	bTrackBuild		: BOOL;
	StartFromTrack	: I_Track;
	EndAtTrack		: I_Track;
END_VAR
fbR_TrigExecute(CLK := bExecute);
IF fbR_TrigExecute.Q AND NOT bBusy THEN
	nState := 10;
	bBusy := TRUE;
	bError := FALSE;
END_IF


CASE nState OF 

	10:	// Init Track-Table
	
		// *******************************************************************
		// *** This code must be eddited according to machine/track layout ***
		// *******************************************************************
	
		nStartFromTrack	:= 0;		// 0 for the first track all others according to their predecessor!
	    	nEndAtTrack := 0;		// 0 for the first track all others according to their successor! 		
		     bCloseLoop := FALSE;	// TRUE for circular track	
			
			
		TrackTable[1,1] :=   0.0;	// x-koordinate
		TrackTable[1,2] :=   0.0;	// y-koordinate
		TrackTable[1,3] :=   0.0;	// c
		
		TrackTable[2,1] :=   0.0;	// x-koordinate
		TrackTable[2,2] :=   0.0;	// y-koordinate
		TrackTable[2,3] :=   0.0;	// c		
		
		TrackTable[3,1] :=   0.0;	// x-koordinate
		TrackTable[3,2] :=   0.0;	// y-koordinate
		TrackTable[3,3] :=   0.0;	// c		
	
		TrackTable[4,1] :=   0.0;	// x-koordinate
		TrackTable[4,2] :=   0.0;	// y-koordinate
		TrackTable[4,3] :=   0.0;	// c		
	
		TrackTable[5,1] :=   0.0;	// x-koordinate
		TrackTable[5,2] :=   0.0;	// y-koordinate
		TrackTable[5,3] :=   0.0;	// c		
	
		TrackTable[6,1] :=   0.0;	// x-koordinate
		TrackTable[6,2] :=   0.0;	// y-koordinate
		TrackTable[6,3] :=   0.0;	// c				
		
		nState := 20;
		
		
	20:	// Building the track
		IF nStartFromTrack > 0 THEN
			StartFromTrack := ipTrack[nStartFromTrack];
		END_IF
		
		IF nEndAtTrack > 0 THEN
			EndAtTrack := ipTrack[nStartFromTrack];
		END_IF

		bTrackBuild := FALSE;
		IF  nStartFromTrack > 0 
		AND     nEndAtTrack > 0
		THEN
			IF fbTrackStandard.BuildTrack(TrackTable, StartFromTrack.std, EndAtTrack.std, bCloseLoop) THEN
				bTrackBuild := TRUE;
			END_IF
		ELSIF nStartFromTrack > 0 THEN
			IF fbTrackStandard.BuildTrack(TrackTable, StartFromTrack.std, 0, bCloseLoop) THEN
				bTrackBuild := TRUE;
			END_IF
		ELSIF nEndAtTrack > 0 THEN
			IF fbTrackStandard.BuildTrack(TrackTable, 0, EndAtTrack.std, bCloseLoop) THEN
				bTrackBuild := TRUE;
			END_IF
		ELSE
			IF fbTrackStandard.BuildTrack(TrackTable, 0, 0, bCloseLoop) THEN
				bTrackBuild := TRUE;
			END_IF			
		END_IF
		
		IF bTrackBuild THEN
			nState := 30;	
		END_IF
	
		
	30: 	
		IF fbTrackStandard.P_BuildTrack.Done THEN
			nState := 100;
		END_IF
		
					 
	100: 	// Track build done
			fTrackLength := fbTrackStandard.GetLength();
				   bBusy := FALSE;
			  Initialize := TRUE;
			
			IF NOT bExecute THEN
				Initialize := FALSE;
				    nState := 0;
			END_IF
	
END_CASE
END_METHOD

END_FUNCTION_BLOCK

// ---- 1_Industry/VISUs/OperationalControlPad.TcVIS
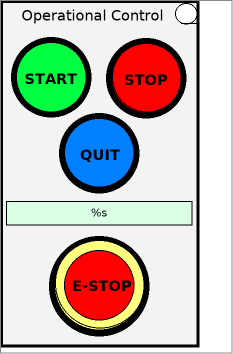
VISUALIZATION OperationalControlPad  // 233x354
VAR_IN_OUT
	stVisOperationalControl	: ST_Vis_OperationalControl;
END_VAR
    Rectangle (0,0 199x347)
    Label (9,1 167x29), "Operational Control"
    Ellipse (11,37 80x80)
    Ellipse (16,42 70x70)
    Ellipse (16,42 70x70), invisible if: NOT stVisOperationalControl.bStartButtonLamp
    Ellipse (106,38 80x80)
    Ellipse (111,43 70x70)
    Ellipse (111,43 70x70), invisible if: Not stVisOperationalControl.bStopButtonLamp
    Ellipse (59,113 80x80)
    Ellipse (64,118 70x70)
    Ellipse (64,118 70x70), invisible if: NOT stVisOperationalControl.bQuitButtonLamp
    Label (13,64 76x30), "START"
    Label (108,65 76x30), "STOP"
    Label (62,140 76x30), "QUIT"
    Rectangle (6,201 186x24), "%s", text variable: stVisOperationalControl.sMessage
    Ellipse (49,236 100x100)
    Ellipse (54,240 90x90)
    Ellipse (64,250 70x70)
    Ellipse (64,250 70x70), invisible if: NOT stVisOperationalControl.bEStopButtonLamp
    Label (64,271 76x30), "E-STOP"
    Rectangle (6,201 186x24), "%s", text variable: stVisOperationalControl.sMessage, invisible if: NOT stVisOperationalControl.bMessageColorRed
    Rectangle (6,201 186x24), "%s", text variable: stVisOperationalControl.sMessage, invisible if: NOT stVisOperationalControl.bMessageColorGreen
    Ellipse (16,42 70x70)
        tap stVisOperationalControl.bStartButtunState
    Ellipse (112,42 70x70)
        tap stVisOperationalControl.bStopButtonState
    Ellipse (64,117 70x70)
        tap stVisOperationalControl.bQuitButtonState
    Ellipse (55,238 90x90)
        toggle stVisOperationalControl.bEStopButtonState
    Ellipse (175,3 22x21)
    Line (218,-7) (233,-6)
    Line (181,23) (197,23)
    Rectangle (158,2 40x30)
        OnMouseClick: execute { stVisOperationalControl.bVisInvisibleButton := TRUE; }
END_VISUALIZATION

// ---- 1_Industry/VISUs/StarterKitStateMachinelPad.TcVIS
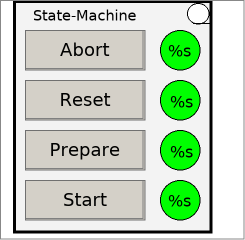
VISUALIZATION StarterKitStateMachinelPad  // 245x240
VAR_IN_OUT
	
	stControlPadControl		:   ST_Vis_ControlPadControl;

END_VAR
    Rectangle (13,0 199x233)
    Button (25,30 120x40), "Abort"
        tap stControlPadControl.bButtonState_Abort p3779583253=TRUE
    Button (25,80 120x40), "Reset"
        tap stControlPadControl.bButtonState_Reset
    Button (25,130 120x40), "Prepare"
        tap stControlPadControl.bButtonState_Prepare
    Button (25,180 120x40), "Start"
        tap stControlPadControl.bButtonState_Start
    Ellipse (160,30 40x40)
    Ellipse (160,30 40x40), invisible if: NOT stControlPadControl.bStateSignalAbortYellow
    Group (160,80 40x40)
        Ellipse (0,0 40x40)
        Ellipse (0,0 40x40), invisible if: NOT stControlPadControl.bStateSignalResetYellow
        Ellipse (0,0 40x40), invisible if: NOT stControlPadControl.bStateSignalResetGreen
    Group (160,130 40x40)
        Ellipse (0,0 40x40)
        Ellipse (0,0 40x40), invisible if: NOT stControlPadControl.bStateSignalPrepareYellow
        Ellipse (0,0 40x40), invisible if: NOT stControlPadControl.bStateSignalPrepareGreen
    Group (160,180 40x40)
        Ellipse (0,0 40x40)
        Ellipse (0,0 40x40), invisible if: NOT stControlPadControl.bStateSignalExecuteYellow
        Ellipse (0,0 40x40), invisible if: NOT stControlPadControl.bStateSignalExecuteGreen
    Ellipse (160,30 40x40), invisible if: NOT stControlPadControl.bStateSignalAbortBlue
    Ellipse (160,30 40x40), invisible if: NOT stControlPadControl.bStateSignalAbortGreen
    Label (19,1 132x29), "State-Machine"
    Textfield (159,35 42x32), "%s", text variable: stControlPadControl.iAbortSequenceState, invisible if: stControlPadControl.bAbortSequenceStateInvisible
    Textfield (161,86 42x32), "%s", text variable: stControlPadControl.iResetSequenceState, invisible if: stControlPadControl.bResetSequenceStateInvisible
    Textfield (161,136 42x32), "%s", text variable: stControlPadControl.iPrepareSequenceState, invisible if: stControlPadControl.bPrepareSequenceStateInvisible
    Textfield (159,185 42x32), "%s", text variable: stControlPadControl.iStartSequenceState, invisible if: stControlPadControl.bStartSequenceStateInvisible
    Ellipse (187,3 22x21)
    Line (230,-7) (245,-6)
    Line (193,23) (209,23)
    Rectangle (179,3 32x25)
        OnMouseClick: execute { stControlPadControl.bVisInvisibleButton := TRUE; }
END_VISUALIZATION

// ---- GlobalTextList.TcGTLO
TEXTLIST GlobalTextList
  632 = '\txPlanar'
  135 = '\tXPlanar'
  427 = '\nGroup\nNotReady'
  425 = '\nGroup\nStandby'
  140 = '%.3f'
  243 = '%d'
  602 = '%d /'
  145 = '%d Axes'
  43 = '%s'
  245 = '+'
  246 = '-'
  532 = '/'
  81 = '1'
  902 = '2'
  489 = '3'
  115 = '4'
  268 = '5'
  274 = 'A'
  39 = 'Abort'
  56 = 'Activated'
  726 = 'Activating'
  774 = 'ActivationState'
  215 = 'B'
  306 = 'Busy'
  671 = 'C'
  224 = 'CA_Group'
  560 = 'E-STOP'
  144 = 'Enable Requested FALSE'
  143 = 'Enable Requested TRUE'
  51 = 'Entrance Location'
  790 = 'Error in the Group or in one of the axes'
  789 = 'error on the\ngroup or in one\nof the axes'
  331 = 'Error: %d'
  1811 = 'Exit Location'
  146 = 'General'
  431 = 'Group\nErrorDisabled'
  430 = 'Group\nErrorEnabled'
  429 = 'GroupDisabled'
  428 = 'GroupErrorStop'
  424 = 'GroupMoving'
  426 = 'GroupStopping'
  750 = 'GVL_StationVisu.aMoverInQueue[INDEX]'
  748 = 'GVL_StationVisu.aMoverInSequence[INDEX].nMover'
  749 = 'GVL_StationVisu.aMoverInSequence[INDEX].nSequence'
  413 = 'GVL_XPlanarVisuDiag.aMoverInSequence[INDEX].nMover'
  498 = 'GVL_XPlanarVisuDiag.aMoverInSequence[INDEX].nSequence'
  53 = 'Home'
  152 = 'Inactive'
  142 = 'INVALID'
  938 = 'M1'
  303 = 'M2'
  38 = 'M3'
  609 = 'M4'
  432 = 'MC_AddAxis'
  783 = 'MC_GroupDisable'
  786 = 'MC_GroupEnable'
  784 = 'MC_GroupHalt'
  434 = 'MC_GroupReset'
  785 = 'MC_GroupStop'
  433 = 'MC_RemAxis'
  787 = 'MC_UngroupAllAxes'
  114 = 'Mover'
  348 = 'Mover:'
  522 = 'MoverId:'
  1100 = 'NumMoversReq.'
  788 = 'one axis\nnot ready'
  807 = 'OnTrack'
  105 = 'Operational Control'
  49 = 'Operational Control Pad'
  819 = 'PosA'
  255 = 'PosB'
  653 = 'PosC'
  837 = 'PosX'
  932 = 'PosY'
  30 = 'PosZ'
  953 = 'Prepare'
  927 = 'Process'
  1737 = 'Prozess Location'
  1111 = 'Queue'
  872 = 'Queue Location'
  509 = 'QueueGap'
  675 = 'QueuePositions'
  134 = 'QUIT'
  40 = 'Reset'
  42 = 'Run'
  41 = 'Start'
  678 = 'START'
  260 = 'State'
  390 = 'State-Machine'
  839 = 'State-Machine Pad'
  291 = 'Station'
  197 = 'Station Parameter'
  461 = 'Station: %d'
  1657 = 'Station: %s'
  141 = 'Status'
  939 = 'STOP'
  499 = 'Track'
  900 = 'X'
  313 = 'y'
END_TEXTLIST

// ---- VISUs/CmdHistory/VI_CmdHistorySide.TcVIS
VISUALIZATION VI_CmdHistorySide  // 2x2
END_VISUALIZATION

// ---- VISUs/CmdHistory/VI_CmdHistorySub.TcVIS
VISUALIZATION VI_CmdHistorySub  // 2x2
END_VISUALIZATION

// ---- VISUs/ControlXplanar/VI_Control_Xplanar.TcVIS
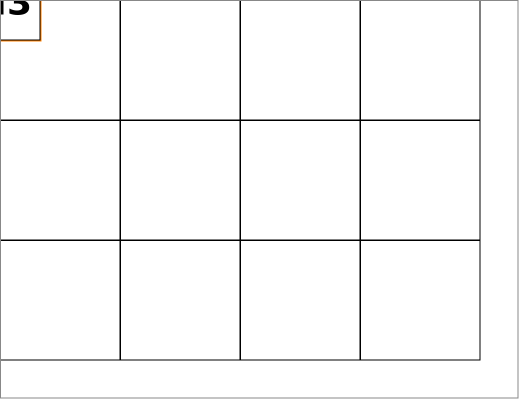
VISUALIZATION VI_Control_Xplanar  // 519x399
    Rectangle (0,0 120x120)
    Rectangle (120,0 120x120)
    Rectangle (240,0 120x120)
    Rectangle (360,0 120x120)
    Rectangle (0,120 120x120)
    Rectangle (120,120 120x120)
    Rectangle (240,120 120x120)
    Rectangle (360,120 120x120)
    Rectangle (0,240 120x120)
    Rectangle (120,240 120x120)
    Rectangle (240,240 120x120)
    Rectangle (360,240 120x120)
    Rectangle (-39,-39 80x80), "1"
        p3560616238: MAIN.fbXMotionUnit.fbStation_01_Process.VisuPosX/2
        p2738717112: (720-MAIN.fbXMotionUnit.fbStation_01_Process.VisuPosY)/2
    Rectangle (-39,-39 80x80), "2"
        p3560616238: MAIN.fbXMotionUnit.fbStation_02_Process.VisuPosX/2
        p2738717112: (720-MAIN.fbXMotionUnit.fbStation_02_Process.VisuPosY)/2
    Rectangle (-39,-39 80x80), "3"
        p3560616238: MAIN.fbXMotionUnit.fbStation_03_Process.VisuPosX/2
        p2738717112: (720-MAIN.fbXMotionUnit.fbStation_03_Process.VisuPosY)/2
    Rectangle (-39,-39 80x80), "4"
        p3560616238: MAIN.fbXMotionUnit.fbStation_04_Switch.VisuPosX/2
        p2738717112: (720-MAIN.fbXMotionUnit.fbStation_04_Switch.VisuPosY)/2
    Rectangle (-39,-39 80x80), "5"
        p3560616238: MAIN.fbXMotionUnit.fbStation_05_Switch.VisuPosX/2
        p2738717112: (720-MAIN.fbXMotionUnit.fbStation_05_Switch.VisuPosY)/2
    Rectangle (-37,-37 77x77), "M1"
        p3560616238: MAIN.fbXMotionUnit.fbMover[1].VisuPos.x/2
        p2738717112: (720-MAIN.fbXMotionUnit.fbMover[1].VisuPos.y)/2
    Rectangle (-37,-37 77x77), "M2"
        p3560616238: MAIN.fbXMotionUnit.fbMover[2].VisuPos.x/2
        p2738717112: (720-MAIN.fbXMotionUnit.fbMover[2].VisuPos.y)/2
    Rectangle (-37,-37 77x77), "M4"
        p3560616238: MAIN.fbXMotionUnit.fbMover[4].VisuPos.x/2
        p2738717112: (720-MAIN.fbXMotionUnit.fbMover[4].VisuPos.y)/2
    Rectangle (-37,-37 77x77), "M3"
        p3560616238: MAIN.fbXMotionUnit.fbMover[3].VisuPos.x/2
        p2738717112: (720-MAIN.fbXMotionUnit.fbMover[3].VisuPos.y)/2
END_VISUALIZATION

// ---- VISUs/Helper/VI_NumberHollow.TcVIS
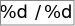
VISUALIZATION VI_NumberHollow  // 75x26
VAR_IN_OUT
	nNumberToDisplay : INT;
	nMaxNumberToDisplay : INT;
END_VAR
    Rectangle (-3,0 34x24), "%d", text variable: nNumberToDisplay
    Rectangle (41,0 32x24), "%d", text variable: nMaxNumberToDisplay
    Rectangle (27,0 17x24), "/", text variable: GVL_XtsVisuLib.nXtsIdMaxToDisplay
END_VISUALIZATION

// ---- VISUs/Helper/VI_NumberSub.TcVIS
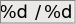
VISUALIZATION VI_NumberSub  // 76x24
VAR_IN_OUT
	nNumberToDisplay : INT;
	nMaxNumberToDisplay : INT;
END_VAR
    Rectangle (-3,0 34x24), "%d", text variable: nNumberToDisplay
    Rectangle (41,0 32x24), "%d", text variable: nMaxNumberToDisplay
    Rectangle (27,0 17x24), "/"
END_VISUALIZATION

// ---- VISUs/Station/VI_Station.TcVIS
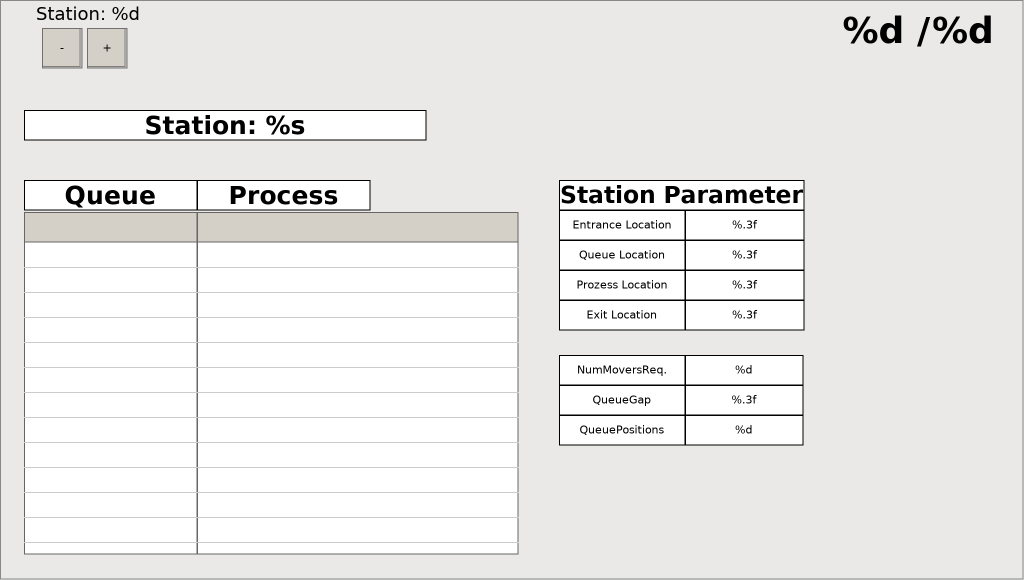
VISUALIZATION VI_Station  // 1024x580
    Frame (0,80 1024x500)
        shows VI_StationSub()
    Rectangle (929,5 77x51), "%d", text variable: GVL_XPlanarVisuDiag.nMaxStationToDisplay
    Rectangle (830,5 103x51), "%d /", text variable: GVL_XPlanarVisuDiag.nStationIdToDisplay
    Button (87,28 40x40), "+", invisible if: GVL_StationVisu.bStationNextInvisible
        tap GVL_XPlanarVisuDiag.bStationNext p1329445385=TRUE
    Button (42,28 40x40), "-", invisible if: GVL_XPlanarVisuDiag.bSationPreviousInvisible
        tap GVL_XPlanarVisuDiag.bStationPrevious
    Rectangle (34,2 108x24), "Station: %d", text variable: GVL_XPlanarVisuDiag.nStationIdToDisplay
END_VISUALIZATION

// ---- VISUs/Station/VI_StationSub.TcVIS
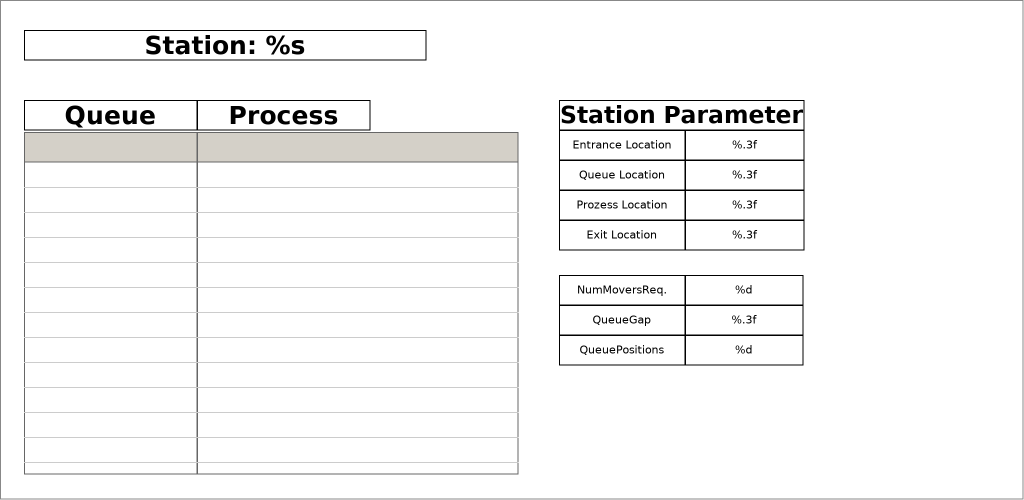
VISUALIZATION VI_StationSub  // 1024x500
    Rectangle (24,30 402x30), "Station: %s", text variable: GVL_XPlanarVisuDiag.sStationName
    Rectangle (24,100 173x30), "Queue"
    Rectangle (197,100 173x30), "Process"
    Table (197,132 321x342), data array: GVL_StationVisu.aMoverInSequence
        p1128707560: GVL_XPlanarVisuDiag.gcnMaxMoverInStation
        p3854506369: GVL_StationVisu.aMoverInSequence[INDEX].nMover
        p1892666644: GVL_StationVisu.aMoverInSequence[INDEX].nSequence
        p2232123230: GVL_XPlanarVisuDiag.aMoverInSequence[INDEX].nMover
        p511219082: GVL_XPlanarVisuDiag.aMoverInSequence[INDEX].nSequence
    Table (24,132 173x342), data array: GVL_XPlanarVisuDiag.aMoverInQueue
        p1128707560: GVL_XPlanarVisuDiag.gcnMaxMoverInStation
        p3854506369: GVL_XPlanarVisuDiag.aMoverInQueue[INDEX]
    Rectangle (559,100 245x30), "Station Parameter"
    Rectangle (559,130 126x30), "Entrance Location"
    Rectangle (559,160 126x30), "Queue Location"
    Rectangle (559,190 126x30), "Prozess Location"
    Rectangle (559,220 126x30), "Exit Location"
    Rectangle (559,275 126x30), "NumMoversReq."
    Rectangle (559,305 126x30), "QueueGap"
    Rectangle (559,335 126x30), "QueuePositions"
    Rectangle (685,130 119x30), "%.3f", text variable: GVL_XPlanarVisuDiag.stStationConfig.fEntranceLocation
    Rectangle (685,160 119x30), "%.3f", text variable: GVL_XPlanarVisuDiag.stStationConfig.fQueueLocation
    Rectangle (685,190 119x30), "%.3f", text variable: GVL_XPlanarVisuDiag.stStationConfig.fProzessLocation
    Rectangle (685,220 119x30), "%.3f", text variable: GVL_XPlanarVisuDiag.stStationConfig.fExitLocation
    Rectangle (685,275 118x30), "%d", text variable: GVL_XPlanarVisuDiag.stStationConfig.nNumMoversRequired
    Rectangle (685,305 118x30), "%.3f", text variable: GVL_XPlanarVisuDiag.stStationConfig.fQueueGap
    Rectangle (685,335 118x30), "%d", text variable: GVL_XPlanarVisuDiag.stStationConfig.nNumQueuePositions
END_VISUALIZATION

// ---- VISUs/Visualization.TcVIS
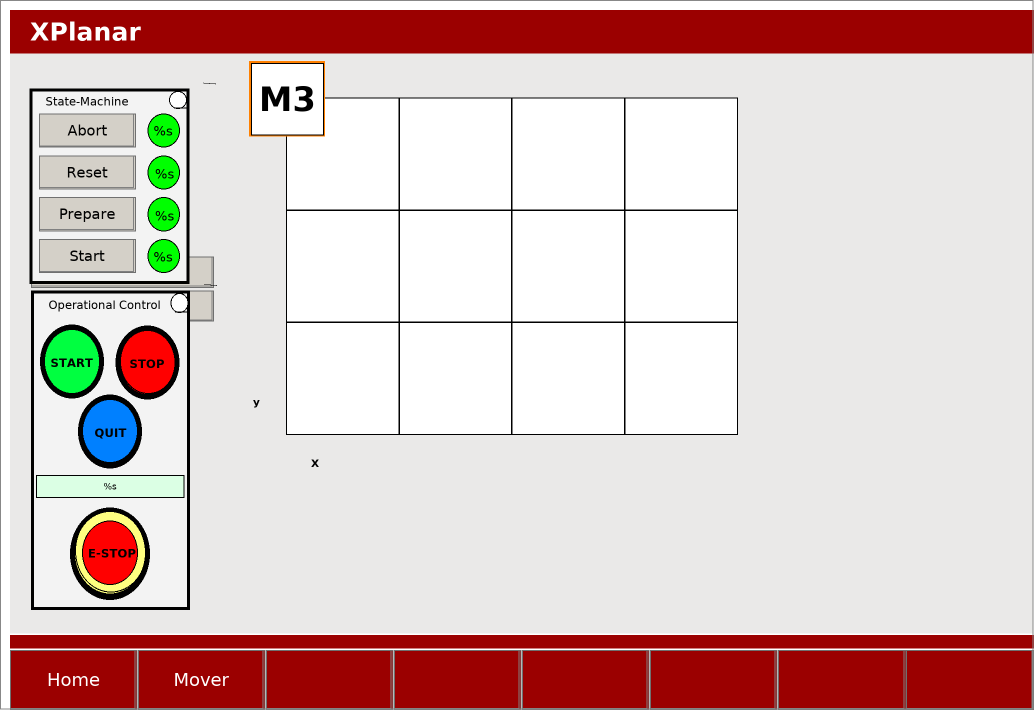
VISUALIZATION Visualization  // 1034x710
    Frame (10,53 1023x580)
        shows VI_MainSide()
        shows Tc3_XPlanarStandard.VI_MoverLogOverview()
        shows VI_EtherCatDiag()
        shows VI_MoverDiag()
        shows VI_MoverTuning()
        shows VI_MoverDiag()
        shows VI_Station()
        p1165984742: GVL_XtsVisu.pGroupRef[1]^.NcToPlc.Common.GroupStatus
        p547225198: GVL_XtsVisu.pGroupRef[1]
    Rectangle (10,10 1024x43), "XPlanar"
    Rectangle (10,635 1024x13)
    Button (10,650 127x60), "Home"
        OnMouseDown: FrameSelectionChange Selection=SelectedFrame=87eec691-4479-469a-bdd2-91ec7a1bb6bd, GlobSel=AssignType=Directly, SelType=Locally
    Button (138,650 127x60), "Mover"
        OnMouseUp: FrameSelectionChange Selection=SelectedFrame=87eec691-4479-469a-bdd2-91ec7a1bb6bd, Selection=1, GlobSel=AssignType=Directly, SelType=Locally
    Button (266,650 127x60)
    Button (394,650 127x60)
    Button (522,650 127x60)
    Button (650,650 127x60)
    Button (906,650 128x60)
    Button (778,650 128x60)
END_VISUALIZATION

// ---- VISUs/Visualization.TcVIS
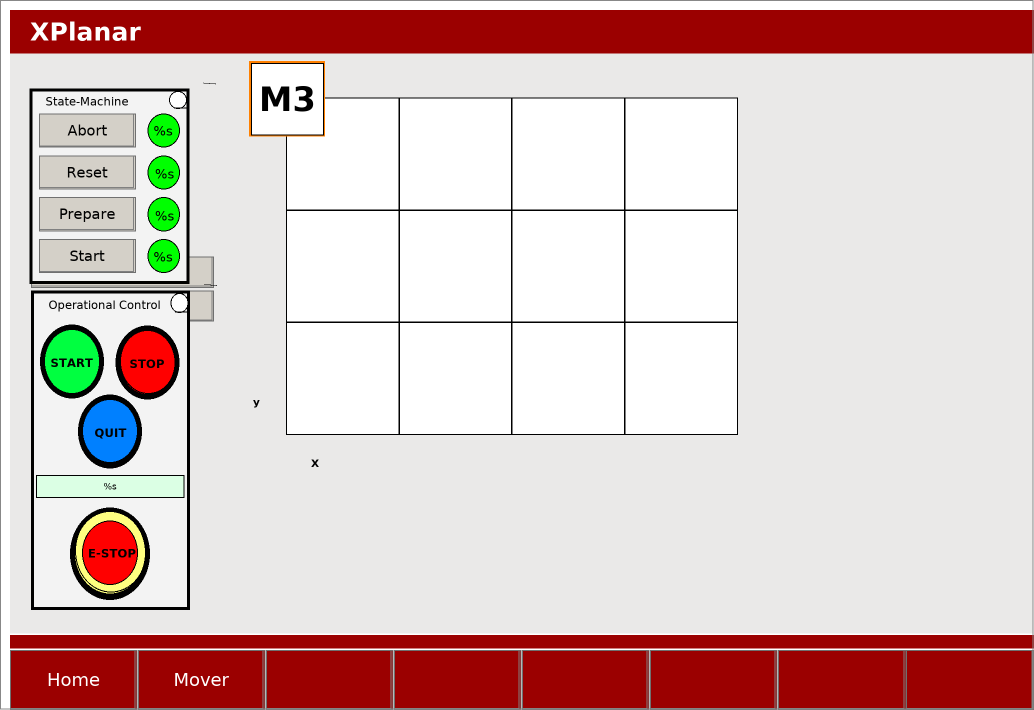
VISUALIZATION Visualization  // 1034x710
    Frame (10,53 1023x580)
        shows VI_MainSide()
        shows Tc3_XPlanarStandard.VI_MoverLogOverview()
        shows VI_EtherCatDiag()
        shows VI_MoverDiag()
        shows VI_MoverTuning()
        shows VI_MoverDiag()
        shows VI_Station()
        p1165984742: GVL_XtsVisu.pGroupRef[1]^.NcToPlc.Common.GroupStatus
        p547225198: GVL_XtsVisu.pGroupRef[1]
    Rectangle (10,10 1024x43), "XPlanar"
    Rectangle (10,635 1024x13)
    Button (10,650 127x60), "Home"
        OnMouseDown: FrameSelectionChange Selection=SelectedFrame=87eec691-4479-469a-bdd2-91ec7a1bb6bd, GlobSel=AssignType=Directly, SelType=Locally
    Button (138,650 127x60), "Mover"
        OnMouseUp: FrameSelectionChange Selection=SelectedFrame=87eec691-4479-469a-bdd2-91ec7a1bb6bd, Selection=1, GlobSel=AssignType=Directly, SelType=Locally
    Button (266,650 127x60)
    Button (394,650 127x60)
    Button (522,650 127x60)
    Button (650,650 127x60)
    Button (906,650 128x60)
    Button (778,650 128x60)
END_VISUALIZATION

// ---- VISUs/VI_MainSide.TcVIS
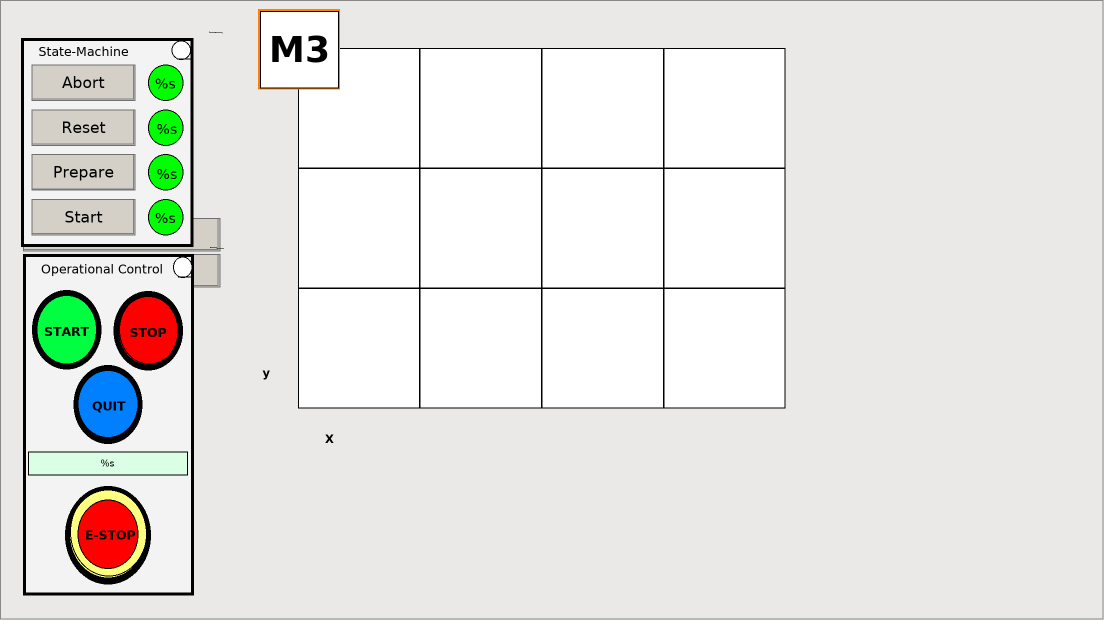
VISUALIZATION VI_MainSide  // 1104x620
    Polygon (172,343) (173,344)
    Frame (298,48 527x399)
        shows VI_Control_Xplanar()
    Label (316,424 27x30), "X"
    Label (253,358 27x30), "y"
    Button (23,254 197x33), "Operational Control Pad", invisible if: NOT stVisControl.stOperatorPad.bVisInvisible
        p3560616238: stVisControl.stOperatorPad.nButtonPositionX
        p2738717112: stVisControl.stOperatorPad.nButtonPositionY
        OnMouseClick: execute { stVisControl.stOperatorPad.bVisInvisibleButton := FALSE; }
    Button (23,218 197x33), "State-Machine Pad", invisible if: NOT stVisControl.stControlPad.bVisInvisible
        p3560616238: stVisControl.stControlPad.nButtonPositionX
        p2738717112: stVisControl.stControlPad.nButtonPositionY
        OnMouseClick: execute { stVisControl.stControlPad.bVisInvisibleButton := FALSE; }
    Frame (10,38 212x215), invisible if: stVisControl.stControlPad.bVisInvisible
        shows StarterKitStateMachinelPad(stControlPadControl := stVisControl.stControlPad)
        p3560616238: stVisControl.stControlPad.nFramePositionX
        p2738717112: stVisControl.stControlPad.nFramePositionY
    Frame (23,254 200x348), invisible if: stVisControl.stOperatorPad.bVisInvisible
        shows OperationalControlPad(stVisOperationalControl := stVisControl.stOperatorPad)
        p3560616238: stVisControl.stOperatorPad.nFramePositionX
        p2738717112: stVisControl.stOperatorPad.nFramePositionY
END_VISUALIZATION

// ---- VISUs/VI_Tc3_XPlanarUtility.TcVIS
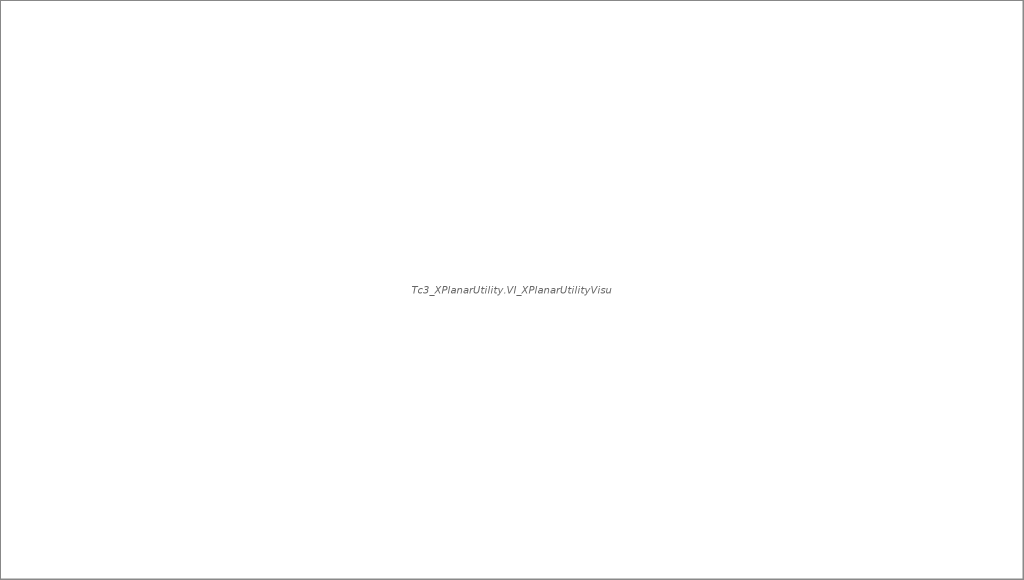
VISUALIZATION VI_Tc3_XPlanarUtility  // 1024x580
    Frame (0,0 1024x580)
        shows Tc3_XPlanarUtility.VI_XPlanarUtilityVisu()
END_VISUALIZATION
